FUNCTION_BLOCK CollectionChangedEventHandler EXTENDS CollectionEventHandler

METHOD PUBLIC HandleEvent
VAR_INPUT
	Event : I_Event;
END_VAR
VAR
	changedEvent : I_CollectionChangedEvent;
END_VAR
IF __QUERYINTERFACE(Event, changedEvent) THEN
	_eventReceived := TRUE;
	fromExpected := changedEvent.Target = expectedOriginator;
END_IF
END_METHOD

END_FUNCTION_BLOCK

(* stored: Version 1.1.0.1, ProductVersion 3.1.4024.12
   POU CollectionChangedEventHandler: Id {624d4e7f-4cae-4871-b4f1-8321a9ffcc81}, SpecialFunc None
   Method HandleEvent: Id {d6b42d48-9627-422d-af26-eee80c59dc1d} *)
